TYPE ST_SlaveState :
STRUCT
	/// slave state 
	eEcState: E_EcCommState;
	nReserved: UINT;
	bError: BOOL;
	bInvalidVPRS: BOOL;
	nReserved2: UINT;
	/// link state 
	bNoCommToSlave: BOOL;
	bLinkError: BOOL;
	bMissingLink: BOOL;
	bUnexpectedLink: BOOL;
	bPortA: BOOL;
	bPortB: BOOL;
	bPortC: BOOL;
	bPortD: BOOL;
END_STRUCT
END_TYPE

(* stored: Version 1.1.0.1, ProductVersion 3.1.0.12
   DUT ST_SlaveState: Id {b576ccdf-3c22-4a33-b427-adf6497f1144} *)
